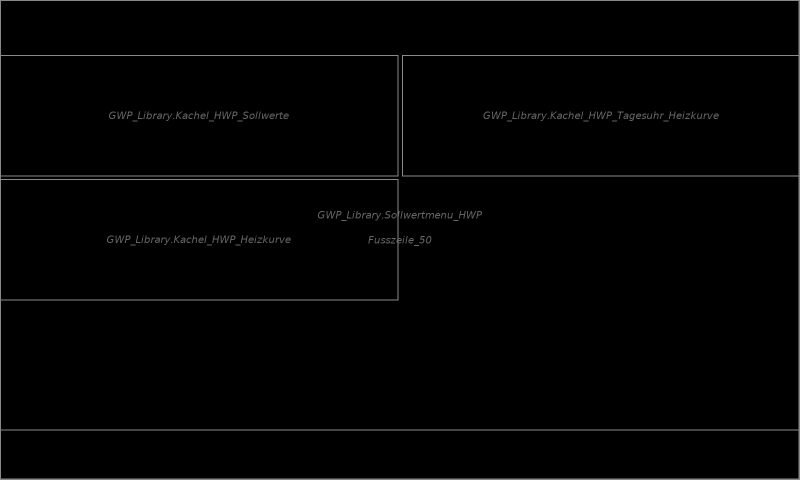
VISUALIZATION Sollwertmenu_HWP  // 800x480
    Frame (0,0 800x430)
        shows GWP_Library.Sollwertmenu_HWP()
    Frame (0,55 398x121)
        shows GWP_Library.Kachel_HWP_Sollwerte(FB_Kreis_3KO := Main.Kreis_3KO_0)
        OnMouseClick: change screen: HWP_SP_Sollwerte
    Frame (402,55 398x121)
        shows GWP_Library.Kachel_HWP_Tagesuhr_Heizkurve()
        OnMouseClick: change screen: HWP_SP_CLK_D
    Frame (0,179 398x121)
        shows GWP_Library.Kachel_HWP_Heizkurve()
        OnMouseClick: change screen: HWP_SP_GR_4_ohne_RE
    Frame (0,0 800x480)
        shows Fusszeile_50()
END_VISUALIZATION

(* stored: Version 1.1.0.1, ProductVersion 3.1.4022.6
   Visu Sollwertmenu_HWP: Id {636a4939-954f-45fd-a001-de97d7490aa6} *)
